INTERFACE ITF_MCMachineControl_HMI_Connector EXTENDS ITF_BaseTopElement_HMI_Connector

END_INTERFACE

(* stored: Version 1.1.0.1
   Itf ITF_MCMachineControl_HMI_Connector: Id {d570e5d8-dcb3-079b-12de-407ccb79a8e5} *)
